// TIA Portal V21 export
DATA_BLOCK "HWData"   // DB3
{ S7_Optimized_Access := 'TRUE' }
// stored: AutoNumber false, MemoryReserve 0
   VAR
      CombiNumber : Int := 0;   // Number according to PLC hardware combination
      ConfigSlots : Array[1.."K_MaxHWCombiNumber"] of "LCC_typeCPUET200SP";   // Slots configurations for all PLC hardware combinations
      CPUET200SP_StatusID : USInt;
      CPUET200SP_Status : DWord;
      CPUET200SP_Config { S7_SetPoint := 'True'} : "LCC_typeCPUET200SP";   // Slots configuration for selected hardware combination
   END_VAR
BEGIN
   ConfigSlots[1].slots[4].actSlotNumber := 132;
   ConfigSlots[1].slots[5].actSlotNumber := 133;
   ConfigSlots[1].slots[6].actSlotNumber := 134;
   ConfigSlots[1].slots[7].actSlotNumber := 7;
   ConfigSlots[1].slots[8].actSlotNumber := 136;
   ConfigSlots[1].slots[9].actSlotNumber := 9;
   ConfigSlots[1].slots[10].actSlotNumber := 10;
   ConfigSlots[1].slots[11].actSlotNumber := 11;
   ConfigSlots[1].slots[12..16].actSlotNumber := 0;
   ConfigSlots[1].slots[17].actSlotNumber := 12;
   ConfigSlots[1].slots[18].actSlotNumber := 13;
   ConfigSlots[1].slots[19].actSlotNumber := 14;
   ConfigSlots[1].slots[20].actSlotNumber := 0;
   ConfigSlots[1].slots[21].actSlotNumber := 15;
   ConfigSlots[2].slots[4].actSlotNumber := 132;
   ConfigSlots[2].slots[5].actSlotNumber := 133;
   ConfigSlots[2].slots[6].actSlotNumber := 134;
   ConfigSlots[2].slots[7].actSlotNumber := 7;
   ConfigSlots[2].slots[8].actSlotNumber := 136;
   ConfigSlots[2].slots[9].actSlotNumber := 9;
   ConfigSlots[2].slots[10].actSlotNumber := 10;
   ConfigSlots[2].slots[11].actSlotNumber := 11;
   ConfigSlots[2].slots[12..14].actSlotNumber := 0;
   ConfigSlots[2].slots[15].actSlotNumber := 12;
   ConfigSlots[2].slots[16].actSlotNumber := 0;
   ConfigSlots[2].slots[17].actSlotNumber := 13;
   ConfigSlots[2].slots[18].actSlotNumber := 14;
   ConfigSlots[2].slots[19].actSlotNumber := 15;
   ConfigSlots[2].slots[20].actSlotNumber := 16;
   ConfigSlots[2].slots[21].actSlotNumber := 17;
   ConfigSlots[3].slots[4].actSlotNumber := 132;
   ConfigSlots[3].slots[5].actSlotNumber := 133;
   ConfigSlots[3].slots[6].actSlotNumber := 134;
   ConfigSlots[3].slots[7].actSlotNumber := 7;
   ConfigSlots[3].slots[8].actSlotNumber := 136;
   ConfigSlots[3].slots[9].actSlotNumber := 9;
   ConfigSlots[3].slots[10].actSlotNumber := 10;
   ConfigSlots[3].slots[11].actSlotNumber := 11;
   ConfigSlots[3].slots[12..15].actSlotNumber := 0;
   ConfigSlots[3].slots[16].actSlotNumber := 12;
   ConfigSlots[3].slots[17].actSlotNumber := 13;
   ConfigSlots[3].slots[18].actSlotNumber := 14;
   ConfigSlots[3].slots[19].actSlotNumber := 15;
   ConfigSlots[3].slots[20].actSlotNumber := 16;
   ConfigSlots[3].slots[21].actSlotNumber := 17;
   ConfigSlots[4].slots[4].actSlotNumber := 132;
   ConfigSlots[4].slots[5].actSlotNumber := 133;
   ConfigSlots[4].slots[6].actSlotNumber := 134;
   ConfigSlots[4].slots[7].actSlotNumber := 7;
   ConfigSlots[4].slots[8].actSlotNumber := 136;
   ConfigSlots[4].slots[9].actSlotNumber := 9;
   ConfigSlots[4].slots[10].actSlotNumber := 10;
   ConfigSlots[4].slots[11].actSlotNumber := 11;
   ConfigSlots[4].slots[12..14].actSlotNumber := 0;
   ConfigSlots[4].slots[15].actSlotNumber := 12;
   ConfigSlots[4].slots[16].actSlotNumber := 13;
   ConfigSlots[4].slots[17].actSlotNumber := 14;
   ConfigSlots[4].slots[18].actSlotNumber := 15;
   ConfigSlots[4].slots[19].actSlotNumber := 16;
   ConfigSlots[4].slots[20].actSlotNumber := 17;
   ConfigSlots[4].slots[21].actSlotNumber := 18;
   ConfigSlots[5].slots[5].actSlotNumber := 133;
   ConfigSlots[5].slots[6].actSlotNumber := 134;
   ConfigSlots[5].slots[7].actSlotNumber := 7;
   ConfigSlots[5].slots[8].actSlotNumber := 136;
   ConfigSlots[5].slots[9].actSlotNumber := 9;
   ConfigSlots[5].slots[10].actSlotNumber := 10;
   ConfigSlots[5].slots[11].actSlotNumber := 11;
   ConfigSlots[5].slots[12].actSlotNumber := 12;
   ConfigSlots[5].slots[13..16].actSlotNumber := 0;
   ConfigSlots[5].slots[17].actSlotNumber := 13;
   ConfigSlots[5].slots[18].actSlotNumber := 14;
   ConfigSlots[5].slots[19].actSlotNumber := 15;
   ConfigSlots[5].slots[20].actSlotNumber := 0;
   ConfigSlots[5].slots[21].actSlotNumber := 16;
   ConfigSlots[6].slots[5].actSlotNumber := 133;
   ConfigSlots[6].slots[6].actSlotNumber := 134;
   ConfigSlots[6].slots[7].actSlotNumber := 7;
   ConfigSlots[6].slots[8].actSlotNumber := 136;
   ConfigSlots[6].slots[9].actSlotNumber := 9;
   ConfigSlots[6].slots[10].actSlotNumber := 10;
   ConfigSlots[6].slots[11].actSlotNumber := 11;
   ConfigSlots[6].slots[12].actSlotNumber := 12;
   ConfigSlots[6].slots[13..14].actSlotNumber := 0;
   ConfigSlots[6].slots[15].actSlotNumber := 13;
   ConfigSlots[6].slots[16].actSlotNumber := 0;
   ConfigSlots[6].slots[17].actSlotNumber := 14;
   ConfigSlots[6].slots[18].actSlotNumber := 15;
   ConfigSlots[6].slots[19].actSlotNumber := 16;
   ConfigSlots[6].slots[20].actSlotNumber := 17;
   ConfigSlots[6].slots[21].actSlotNumber := 18;
   ConfigSlots[7].slots[5].actSlotNumber := 133;
   ConfigSlots[7].slots[6].actSlotNumber := 134;
   ConfigSlots[7].slots[7].actSlotNumber := 7;
   ConfigSlots[7].slots[8].actSlotNumber := 136;
   ConfigSlots[7].slots[9].actSlotNumber := 9;
   ConfigSlots[7].slots[10].actSlotNumber := 10;
   ConfigSlots[7].slots[11].actSlotNumber := 11;
   ConfigSlots[7].slots[12].actSlotNumber := 12;
   ConfigSlots[7].slots[13..15].actSlotNumber := 0;
   ConfigSlots[7].slots[16].actSlotNumber := 13;
   ConfigSlots[7].slots[17].actSlotNumber := 14;
   ConfigSlots[7].slots[18].actSlotNumber := 15;
   ConfigSlots[7].slots[19].actSlotNumber := 16;
   ConfigSlots[7].slots[20].actSlotNumber := 17;
   ConfigSlots[7].slots[21].actSlotNumber := 18;
   ConfigSlots[8].slots[5].actSlotNumber := 133;
   ConfigSlots[8].slots[6].actSlotNumber := 134;
   ConfigSlots[8].slots[7].actSlotNumber := 7;
   ConfigSlots[8].slots[8].actSlotNumber := 136;
   ConfigSlots[8].slots[9].actSlotNumber := 9;
   ConfigSlots[8].slots[10].actSlotNumber := 10;
   ConfigSlots[8].slots[11].actSlotNumber := 11;
   ConfigSlots[8].slots[12].actSlotNumber := 12;
   ConfigSlots[8].slots[13..14].actSlotNumber := 0;
   ConfigSlots[8].slots[15].actSlotNumber := 13;
   ConfigSlots[8].slots[16].actSlotNumber := 14;
   ConfigSlots[8].slots[17].actSlotNumber := 15;
   ConfigSlots[8].slots[18].actSlotNumber := 16;
   ConfigSlots[8].slots[19].actSlotNumber := 17;
   ConfigSlots[8].slots[20].actSlotNumber := 18;
   ConfigSlots[8].slots[21].actSlotNumber := 19;
   ConfigSlots[9].slots[6].actSlotNumber := 134;
   ConfigSlots[9].slots[7].actSlotNumber := 7;
   ConfigSlots[9].slots[8].actSlotNumber := 8;
   ConfigSlots[9].slots[9].actSlotNumber := 9;
   ConfigSlots[9].slots[10].actSlotNumber := 10;
   ConfigSlots[9].slots[11].actSlotNumber := 11;
   ConfigSlots[9].slots[12].actSlotNumber := 12;
   ConfigSlots[9].slots[13].actSlotNumber := 13;
   ConfigSlots[9].slots[14..16].actSlotNumber := 0;
   ConfigSlots[9].slots[17].actSlotNumber := 14;
   ConfigSlots[9].slots[18].actSlotNumber := 15;
   ConfigSlots[9].slots[19].actSlotNumber := 16;
   ConfigSlots[9].slots[20].actSlotNumber := 0;
   ConfigSlots[9].slots[21].actSlotNumber := 17;
   ConfigSlots[10].slots[6].actSlotNumber := 134;
   ConfigSlots[10].slots[7].actSlotNumber := 7;
   ConfigSlots[10].slots[8].actSlotNumber := 8;
   ConfigSlots[10].slots[9].actSlotNumber := 9;
   ConfigSlots[10].slots[10].actSlotNumber := 10;
   ConfigSlots[10].slots[11].actSlotNumber := 11;
   ConfigSlots[10].slots[12].actSlotNumber := 12;
   ConfigSlots[10].slots[13].actSlotNumber := 13;
   ConfigSlots[10].slots[14].actSlotNumber := 0;
   ConfigSlots[10].slots[15].actSlotNumber := 14;
   ConfigSlots[10].slots[16].actSlotNumber := 0;
   ConfigSlots[10].slots[17].actSlotNumber := 15;
   ConfigSlots[10].slots[18].actSlotNumber := 16;
   ConfigSlots[10].slots[19].actSlotNumber := 17;
   ConfigSlots[10].slots[20].actSlotNumber := 18;
   ConfigSlots[10].slots[21].actSlotNumber := 19;
   ConfigSlots[11].slots[6].actSlotNumber := 134;
   ConfigSlots[11].slots[7].actSlotNumber := 7;
   ConfigSlots[11].slots[8].actSlotNumber := 8;
   ConfigSlots[11].slots[9].actSlotNumber := 9;
   ConfigSlots[11].slots[10].actSlotNumber := 10;
   ConfigSlots[11].slots[11].actSlotNumber := 11;
   ConfigSlots[11].slots[12].actSlotNumber := 12;
   ConfigSlots[11].slots[13].actSlotNumber := 13;
   ConfigSlots[11].slots[14..15].actSlotNumber := 0;
   ConfigSlots[11].slots[16].actSlotNumber := 14;
   ConfigSlots[11].slots[17].actSlotNumber := 15;
   ConfigSlots[11].slots[18].actSlotNumber := 16;
   ConfigSlots[11].slots[19].actSlotNumber := 17;
   ConfigSlots[11].slots[20].actSlotNumber := 18;
   ConfigSlots[11].slots[21].actSlotNumber := 19;
   ConfigSlots[12].slots[6].actSlotNumber := 134;
   ConfigSlots[12].slots[7].actSlotNumber := 7;
   ConfigSlots[12].slots[8].actSlotNumber := 8;
   ConfigSlots[12].slots[9].actSlotNumber := 9;
   ConfigSlots[12].slots[10].actSlotNumber := 10;
   ConfigSlots[12].slots[11].actSlotNumber := 11;
   ConfigSlots[12].slots[12].actSlotNumber := 12;
   ConfigSlots[12].slots[13].actSlotNumber := 13;
   ConfigSlots[12].slots[14].actSlotNumber := 0;
   ConfigSlots[12].slots[15].actSlotNumber := 14;
   ConfigSlots[12].slots[16].actSlotNumber := 15;
   ConfigSlots[12].slots[17].actSlotNumber := 16;
   ConfigSlots[12].slots[18].actSlotNumber := 17;
   ConfigSlots[12].slots[19].actSlotNumber := 18;
   ConfigSlots[12].slots[20].actSlotNumber := 19;
   ConfigSlots[12].slots[21].actSlotNumber := 20;
   ConfigSlots[13].slots[8].actSlotNumber := 8;
   ConfigSlots[13].slots[9].actSlotNumber := 9;
   ConfigSlots[13].slots[10].actSlotNumber := 10;
   ConfigSlots[13].slots[11].actSlotNumber := 11;
   ConfigSlots[13].slots[12].actSlotNumber := 12;
   ConfigSlots[13].slots[13].actSlotNumber := 13;
   ConfigSlots[13].slots[14].actSlotNumber := 14;
   ConfigSlots[13].slots[15..16].actSlotNumber := 0;
   ConfigSlots[13].slots[17].actSlotNumber := 15;
   ConfigSlots[13].slots[18].actSlotNumber := 16;
   ConfigSlots[13].slots[19].actSlotNumber := 17;
   ConfigSlots[13].slots[20].actSlotNumber := 0;
   ConfigSlots[13].slots[21].actSlotNumber := 18;
   ConfigSlots[14].slots[9].actSlotNumber := 9;
   ConfigSlots[14].slots[10].actSlotNumber := 10;
   ConfigSlots[14].slots[11].actSlotNumber := 11;
   ConfigSlots[14].slots[12].actSlotNumber := 12;
   ConfigSlots[14].slots[13].actSlotNumber := 13;
   ConfigSlots[14].slots[14].actSlotNumber := 14;
   ConfigSlots[14].slots[15].actSlotNumber := 15;
   ConfigSlots[14].slots[16].actSlotNumber := 0;
   ConfigSlots[14].slots[17].actSlotNumber := 16;
   ConfigSlots[14].slots[18].actSlotNumber := 17;
   ConfigSlots[14].slots[19].actSlotNumber := 18;
   ConfigSlots[14].slots[20].actSlotNumber := 19;
   ConfigSlots[14].slots[21].actSlotNumber := 20;
   ConfigSlots[15].slots[8].actSlotNumber := 8;
   ConfigSlots[15].slots[9].actSlotNumber := 9;
   ConfigSlots[15].slots[10].actSlotNumber := 10;
   ConfigSlots[15].slots[11].actSlotNumber := 11;
   ConfigSlots[15].slots[12].actSlotNumber := 12;
   ConfigSlots[15].slots[13].actSlotNumber := 13;
   ConfigSlots[15].slots[14].actSlotNumber := 14;
   ConfigSlots[15].slots[15].actSlotNumber := 0;
   ConfigSlots[15].slots[16].actSlotNumber := 15;
   ConfigSlots[15].slots[17].actSlotNumber := 16;
   ConfigSlots[15].slots[18].actSlotNumber := 17;
   ConfigSlots[15].slots[19].actSlotNumber := 18;
   ConfigSlots[15].slots[20].actSlotNumber := 19;
   ConfigSlots[15].slots[21].actSlotNumber := 20;
   ConfigSlots[16].slots[21].actSlotNumber := 21;
   ConfigSlots[1].slots[2].slotProperty := 1;
   ConfigSlots[1].slots[4..6].slotProperty := 0;
END_DATA_BLOCK
